// TIA Portal V17 export
// export: Created 2022-07-28T18:03:17.581728Z, ExportSetting None, DisplayName Totally Integrated Automation Portal, DisplayVersion V17, DisplayName TIA Portal Openness, DisplayVersion V17, DisplayName TIA Portal Teamcenter Gateway, DisplayVersion V17, DisplayName TIA Portal Version Control Interface, DisplayVersion V17, DisplayName TIA Portal Test Suite Advanced, DisplayVersion V17, DisplayName SINAMICS Startdrive Advanced, DisplayVersion V17, DisplayName SINAMICS DCC, DisplayVersion V17, DisplayName SINAMICS Startdrive G130, G150, S120, S150, SINAMICS MV, S210, DisplayVersion V17, DisplayName SINAMICS Startdrive G110M, G120, G120C, G120D, G120P, G115D, DisplayVersion V17, DisplayName STEP 7 Professional, DisplayVersion V17, DisplayName SIMATIC Energy Suite, DisplayVersion V17, DisplayName STEP 7 CFC, DisplayVersion V17, DisplayName STEP 7 Safety, DisplayVersion V17, DisplayName WinCC Advanced / Unified PC, DisplayVersion V17, DisplayName SIMATIC Visualization Architect, DisplayVersion V17
TYPE "Lib_PLC_PLS"
   STRUCT
      P100MS : Bool;   // 100 мс
      P200MS : Bool;   // 200 мс
      P500MS : Bool;   // 500 мс
      P1S : Bool;   // 1 с
      P2S : Bool;   // 2 с
      P5S : Bool;   // 5 с
      P10S : Bool;   // 10 с
      P60S : Bool;   // 1 хв
      M1S : Bool;   // меандр з періодом 1 с (0.5 с + 0.5 с)
      M2S : Bool;   // меандр з періодом 2 с (1 с + 1 с)
      FirstScan : Bool;   // =1 – перший скан
      b11 : Bool;
      NEWMIN : Bool;   // =1 (на один цикл основної задачі) – початок хвилини
      NEWHR : Bool;   // =1 (на один цикл основної задачі) – початок години
      NEWDAY : Bool;   // =1 (на один цикл основної задачі) – початок доби
      NEWSHIFT : Bool;   // =1 (на один цикл основної задачі) – початок зміни
   END_STRUCT;
END_TYPE
